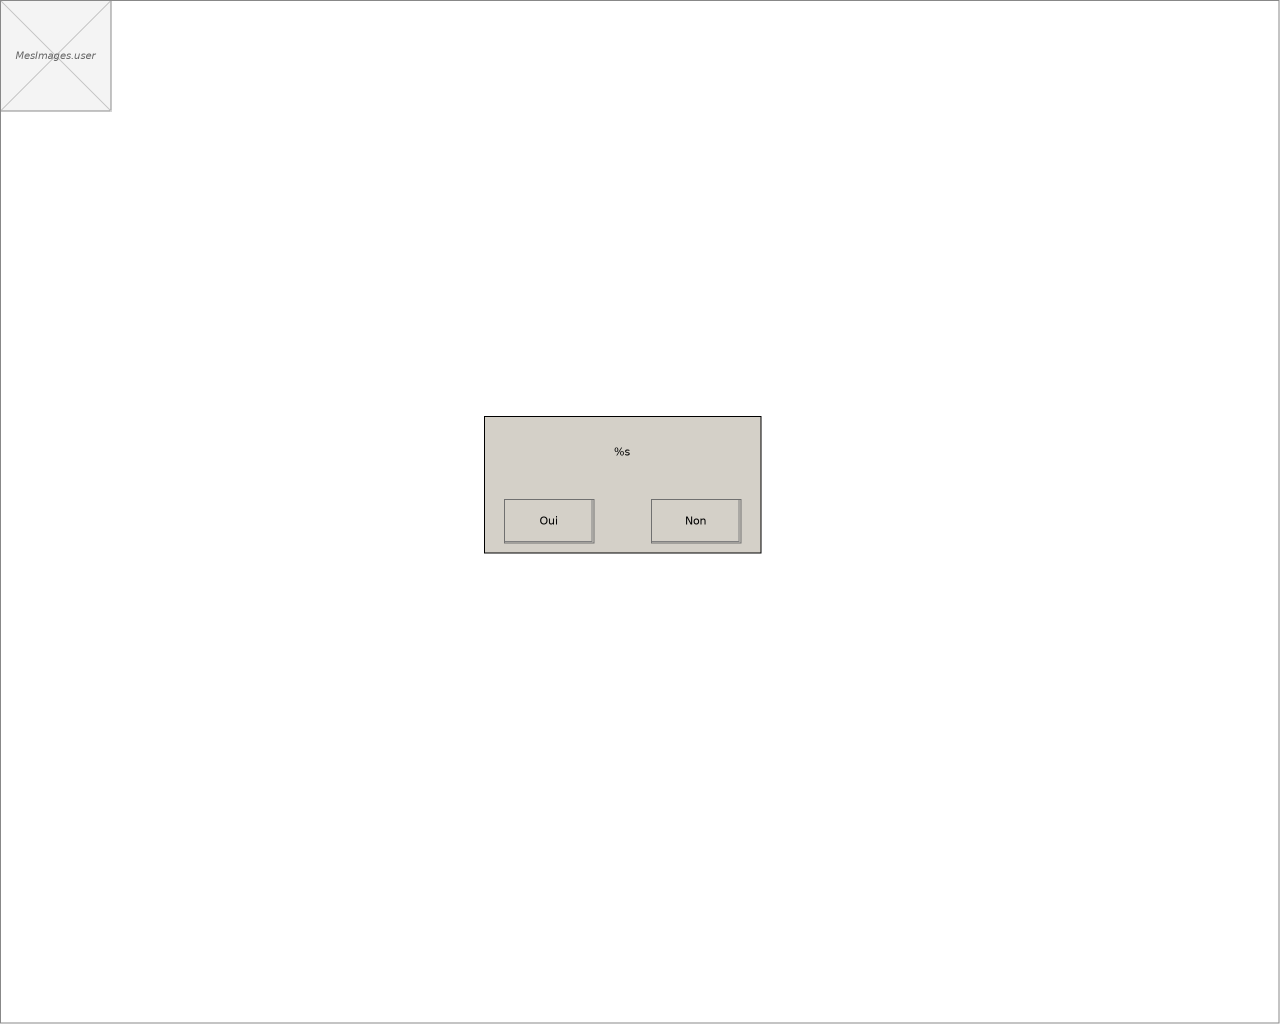
VISUALIZATION UTIL_DELOG  // 1280x1024
    Image (0,0 111x111), image: MesImages.user
    RoundedRectangle (484,416 277x137)
    Textfield (503,422 238x60), "%s", text list: 'TextList_Users_Menu', text index: 3
    Button (504,499 90x44), "Oui"
        toggle PRG_USER.DD_DELOG
        OnMouseClick: change screen: UTIL_MENU
    Button (651,499 90x44), "Non"
        OnMouseClick: change screen: UTIL_MENU
END_VISUALIZATION

(* stored: Version 1.1.0.1, ProductVersion 3.1.4024.10
   Visu UTIL_DELOG: Id {72d42083-9e12-46f3-a0bf-f0ee3c43e96d} *)
